// TwinCAT 3 PLC project TcUnitSample01
// ProgramVersion: 3.1.4022.1
// libraries:
//   Tc2_Standard, * (Beckhoff Automation GmbH)
//   Tc2_System, * (Beckhoff Automation GmbH)
//   Tc2_Utilities, * (Beckhoff Automation GmbH)
//   Tc3_Module, * (Beckhoff Automation GmbH)
//   TcUnit, * (TcUnit)
// project tree:
//   / PlcTask.TcTTO
//   POUs/ FB_Foo.TcPOU, MAIN.TcPOU
//   POUs/TcUnit_Tests/ FB_Foo_Tests.TcPOU, P_Unit_Tests.TcPOU
// real-time tasks:
//   TASK PlcTask: cycle T#10ms, priority 20, ADS port 350

CONFIGURATION TcUnitSample01
    RESOURCE PLC ON TwinCAT3
        TASK PlcTask(INTERVAL := T#10ms, PRIORITY := 20);
        PROGRAM MAIN WITH PlcTask : MAIN;
    END_RESOURCE
END_CONFIGURATION

// ---- POUs/MAIN.TcPOU
PROGRAM MAIN
VAR
END_VAR

P_Unit_Tests();

END_PROGRAM

// ---- POUs/TcUnit_Tests/P_Unit_Tests.TcPOU
PROGRAM P_Unit_Tests
VAR
	fbFoo_Tests		:	FB_Foo_Tests;	
END_VAR

fbFoo_Tests();

END_PROGRAM

// ---- POUs/TcUnit_Tests/FB_Foo_Tests.TcPOU
FUNCTION_BLOCK FB_Foo_Tests
VAR_INPUT
END_VAR
VAR_OUTPUT
	bError			: BOOL;
	bDone			: BOOL;
END_VAR
VAR
	Assert			: FB_ASSERT('FB_Foo');
	tonDelay		: TON;	
	fbFoo_0100		: FB_Foo;
	fbFoo_0200		: FB_Foo;
	fbFoo_0300		: FB_Foo;
	fbFoo_0400		: FB_Foo;	
END_VAR

CASE Assert.State OF
{region "start"}
	16#0000:
		Assert.AbortAfterFail := FALSE;
		Assert.MultipleLog := FALSE;	
		bError := FALSE;
		bDone := FALSE;	
		Assert.State := 16#0100;
{endregion}

{region "Switch_RisingEdgeAndDuration1s_OutIsTrueFor1s"}
	16#0100:
		fbFoo_0100(bSwitch := TRUE, tDuration := T#1S);
		Assert.AreEqualBOOL(TRUE, fbFoo_0100.bOut, 'Switch_RisingEdgeAndDuration1s_OutIsTrueFor1s');
		tonDelay(IN := TRUE, PT := T#900MS);
		IF (tonDelay.Q) THEN
			tonDelay(IN := FALSE);
			Assert.State := 16#0200;
		END_IF	
{endregion}

{region "Switch_RisingEdgeAndDuration1s_OutIsFalseAfter1100ms"}
	16#0200:
		fbFoo_0200(bSwitch := TRUE, tDuration := T#1S);
		tonDelay(IN := TRUE, PT := T#1100MS);
		IF (tonDelay.Q) THEN
			tonDelay(IN := FALSE);
			Assert.AreEqualBOOL(FALSE, fbFoo_0200.bOut, 'Switch_RisingEdgeAndDuration1s_OutIsFalseAfter1100ms');
			Assert.State := 16#0300;
		END_IF	
{endregion}

{region "Switch_RetriggerSwitch_OutKeepsTrue"}
	16#0300:
		fbFoo_0300(bSwitch := TRUE, tDuration := T#500MS);
		Assert.AreEqualBOOL(TRUE, fbFoo_0300.bOut, 'Switch_RetriggerSwitch_OutKeepsTrue');
		tonDelay(IN := TRUE, PT := T#400MS);
		IF (tonDelay.Q) THEN
			tonDelay(IN := FALSE);
			fbFoo_0300(bSwitch := FALSE);
			Assert.State := 16#0310;			
		END_IF		
		
	16#0310:
		fbFoo_0300(bSwitch := TRUE, tDuration := T#500MS);
		Assert.AreEqualBOOL(TRUE, fbFoo_0300.bOut, 'Switch_RetriggerSwitch_OutKeepsTrue');
		tonDelay(IN := TRUE, PT := T#400MS);
		IF (tonDelay.Q) THEN
			tonDelay(IN := FALSE);
			Assert.State := 16#0400;
		END_IF
{endregion}

{region "Off_RisingEdgeAndOutIsTrue_OutIsFalse"}
	16#0400:
		fbFoo_0400(bSwitch := TRUE, tDuration := T#200MS);
		Assert.AreEqualBOOL(TRUE, fbFoo_0400.bOut, 'Off_RisingEdgeAndOutIsTrue_OutIsFalse');
		tonDelay(IN := TRUE, PT := T#100MS);
		IF (tonDelay.Q) THEN
			tonDelay(IN := FALSE);
			fbFoo_0400(bOff := TRUE);
			Assert.AreEqualBOOL(FALSE, fbFoo_0400.bOut, 'Off_RisingEdgeAndOutIsTrue_OutIsFalse');
			Assert.State := 16#FF00;
		END_IF
{endregion}
		
{region "done"}
	16#FF00:
		Assert.PrintPassed('Done');
		Assert.State := 16#FF10;

	16#FF10:
		bDone := TRUE;
		
{endregion}

{region "error"}
	16#FFFF:
		bError := TRUE;
{endregion}
		
	ELSE
		Assert.StateMachineError();
END_CASE

END_FUNCTION_BLOCK

// ---- POUs/FB_Foo.TcPOU
FUNCTION_BLOCK FB_Foo
VAR_INPUT
	bSwitch					:	BOOL;
	bOff					:	BOOL;
	tDuration				:	TIME := T#10S;
END_VAR
VAR_OUTPUT
	bOut					:	BOOL;
END_VAR
VAR
	tonDuration				:	TON;
	rtrigSwitch				:	R_TRIG;
	rtrigOff				:	R_TRIG;
	bStart					:	BOOL;
END_VAR

rtrigSwitch(CLK := bSwitch);
IF (rtrigSwitch.Q) THEN
	bStart := TRUE;
	bOut := TRUE;
	tonDuration(IN := FALSE);
END_IF

rtrigOff(CLK := bOff);
IF (rtrigOff.Q) THEN
	bStart := FALSE;
	bOut := FALSE;
	tonDuration(IN := FALSE);
END_IF

IF (bStart) THEN
	tonDuration(IN := TRUE, PT := tDuration);
	IF (tonDuration.Q) THEN
		tonDuration(IN := FALSE);
		bOut := FALSE;
		bStart := FALSE;
	END_IF
END_IF

END_FUNCTION_BLOCK
